{attribute 'qualified_only'}
VAR_GLOBAL
	VonMatlab		: REAL := 1;
	NachMatlab		: REAL := 1;
END_VAR

(* stored: Version 1.1.0.1, ProductVersion 3.1.4024.10
   GVL AdsVariables: Id {186c5690-a863-4347-bace-605c9d8bf706} *)
